FUNCTION MAX2 : INT
VAR_INPUT
	a : INT;
	b:INT;
END_VAR
VAR_OUTPUT
	c:INT;
	
END_VAR
VAR
END_VAR

IF a >= b THEN
	MAX2 := a;
	c:=a;
ELSE
	MAX2 := b;
	c:=b;
END_IF

END_FUNCTION

(* stored: Version 1.1.0.1, ProductVersion 3.1.4024.16
   POU MAX2: Id {9132d441-4b4f-4efd-9de7-e7fd407a8bbf}, SpecialFunc None *)
